(* Logix 5000 project; controller Google vendor 1 type 14 code 151 rev 31.11; software revision 31.00; part 4 of 6 *)
(* tags used below, declared in another part *)
   Elev_FWD_Delay : TIMER;
   Elev_REV_Delay : TIMER;
   Elev_Slow : BOOL;
   FaultResetDelay : TIMER;
   HMI_AutoMode : BOOL;
   HMI_LiftJogDown : BOOL;
   HMI_LiftJogUp : BOOL;
   HMI_PB_Reset : BOOL;
   Infeed_Active : BOOL;
   Infeed_Clear : BOOL;
   Infeed_Upstream_ProdCode : DINT;
   Infeed_Upstream_ProdName : STRING;
   Infeed_Z1_MinGapTimer : TIMER;
   Infeed_Z3_MinGapTimer : TIMER;
   Infeed_Zone1 : Zone_Data;
   Infeed_Zone1_2_ProdCode : DINT;
   Infeed_Zone1_2_ProdName : STRING;
   Infeed_Zone1_FWD : BOOL;
   Infeed_Zone1_PE : BOOL;
   Infeed_Zone1_ProdCode : DINT;
   Infeed_Zone1_ProdName : STRING;
   Infeed_Zone1_REV : BOOL;
   Infeed_Zone2 : Zone_Data;
   Infeed_Zone2_3_ProdCode : DINT;
   Infeed_Zone2_3_ProdName : STRING;
   Infeed_Zone2_FWD : BOOL;
   Infeed_Zone2_PE : BOOL;
   Infeed_Zone2_ProdCode : DINT;
   Infeed_Zone2_ProdName : STRING;
   Infeed_Zone2_REV : BOOL;
   Infeed_Zone3 : Zone_Data;
   Infeed_Zone3_4_ProdCode : DINT;
   Infeed_Zone3_4_ProdName : STRING;
   Infeed_Zone3_FWD : BOOL;
   Infeed_Zone3_PE : BOOL;
   Infeed_Zone3_ProdCode : DINT;
   Infeed_Zone3_ProdName : STRING;
   Infeed_Zone3_REV : BOOL;
   Infeed_Zone4 : Zone_Data;
   Infeed_Zone4_FWD : BOOL;
   Infeed_Zone4_PE : BOOL;
   Infeed_Zone4_ProdCode : DINT;
   Infeed_Zone4_ProdName : STRING;
   Infeed_Zone4_REV : BOOL;
   Infeed_Zone_Timeout : TIMER[8];
   L1_Clear_Out : BOOL;
   L1_Empty_Delay : TIMER;
   L1_Full_Delay : TIMER;
   L1_Zone1 : Zone_Data;
   L1_Zone1_2_ProdCode : DINT;
   L1_Zone1_2_ProdName : STRING;
   L1_Zone1_FWD : BOOL;
   L1_Zone1_PE : BOOL;
   L1_Zone1_ProdCode : DINT;
   L1_Zone1_ProdName : STRING;
   L1_Zone1_REV : BOOL;
   L1_Zone2 : Zone_Data;
   L1_Zone2_3_ProdCode : DINT;
   L1_Zone2_3_ProdName : STRING;
   L1_Zone2_FWD : BOOL;
   L1_Zone2_PE : BOOL;
   L1_Zone2_ProdCode : DINT;
   L1_Zone2_ProdName : STRING;
   L1_Zone2_REV : BOOL;
   L1_Zone3 : Zone_Data;
   L1_Zone3_4_ProdCode : DINT;
   L1_Zone3_4_ProdName : STRING;
   L1_Zone3_FWD : BOOL;
   L1_Zone3_PE : BOOL;
   L1_Zone3_ProdCode : DINT;
   L1_Zone3_ProdName : STRING;
   L1_Zone3_REV : BOOL;
   L1_Zone4 : End_Zone_Data;
   L1_Zone4_FWD : BOOL;
   L1_Zone4_PE : BOOL;
   L1_Zone4_ProdCode : DINT;
   L1_Zone4_ProdName : STRING;
   L1_Zone4_REV : BOOL;
   L1_Zone_Timeout : TIMER[8];
   L2_Zone1 : Zone_Data;
   L2_Zone1_REV : BOOL;
   L3_Zone1 : Zone_Data;
   L3_Zone1_REV : BOOL;
   L4_Zone1 : Zone_Data;
   L4_Zone1_REV : BOOL;
   L5_Zone1 : Zone_Data;
   L5_Zone1_REV : BOOL;
   Level_1_Empty : BOOL;
   Level_1_Full : BOOL;
   Lift_Alarm : BOOL;
   Lift_Ascend : BOOL;
   Lift_Conv_PE1 : BOOL;
   Lift_Conv_PE2 : BOOL;
   Lift_Current_Level : DINT;
   Lift_Cycle_Counter : COUNTER;
   Lift_Descend : BOOL;
   Lift_FullSpeed : DINT;
   Lift_L1_Slow_Prox : BOOL;
   Lift_L1_Stop_Prox : BOOL;
   Lift_L2_Slow_Prox : BOOL;
   Lift_L2_Stop_Prox : BOOL;
   Lift_L3_Slow_Prox : BOOL;
   Lift_L3_Stop_Prox : BOOL;
   Lift_L4_Slow_Prox : BOOL;
   Lift_L4_Stop_Prox : BOOL;
   Lift_L5_Slow_Prox : BOOL;
   Lift_L5_Stop_Prox : BOOL;
   Lift_Required_Level : DINT;
   Lift_SlowSpeed : DINT;
   Lift_Zone : Lift_Zone_Data;
   Lift_Zone_ProdCode : DINT;
   Lift_Zone_ProdName : STRING;
   Lift_Zone_Timeout : TIMER[2];
   LiftZone_FWD : BOOL;
   LiftZone_REV : BOOL;
   LiftZoneDownstream_ProdCode : DINT;
   LiftZoneDownstream_ProdName : STRING;
   LiftZoneFWD_ResetTimer : TIMER;
   LiftZoneREV_ResetTimer : TIMER;
   LiftZoneUpstream_ProdCode : DINT;
   LiftZoneUpstream_ProdName : STRING;
   ONS : DINT[6];
   Outfeed_Active : BOOL;
   Safety_Relay_Status : BOOL;
   Sort_Number : DINT;
   System : State;
   System_State : DINT;
(* MainProgram, continued *)

ROUTINE R06_Lift_Operation   (* ladder *)
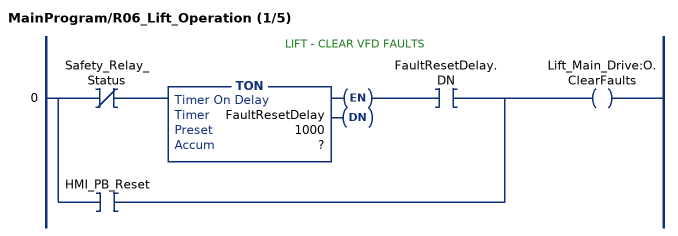
   // LIFT - CLEAR VFD FAULTS
   0: [XIO(Safety_Relay_Status) TON(FaultResetDelay,?,?) XIC(FaultResetDelay.DN) ,XIC(HMI_PB_Reset) ]OTE(Lift_Main_Drive:O.ClearFaults);
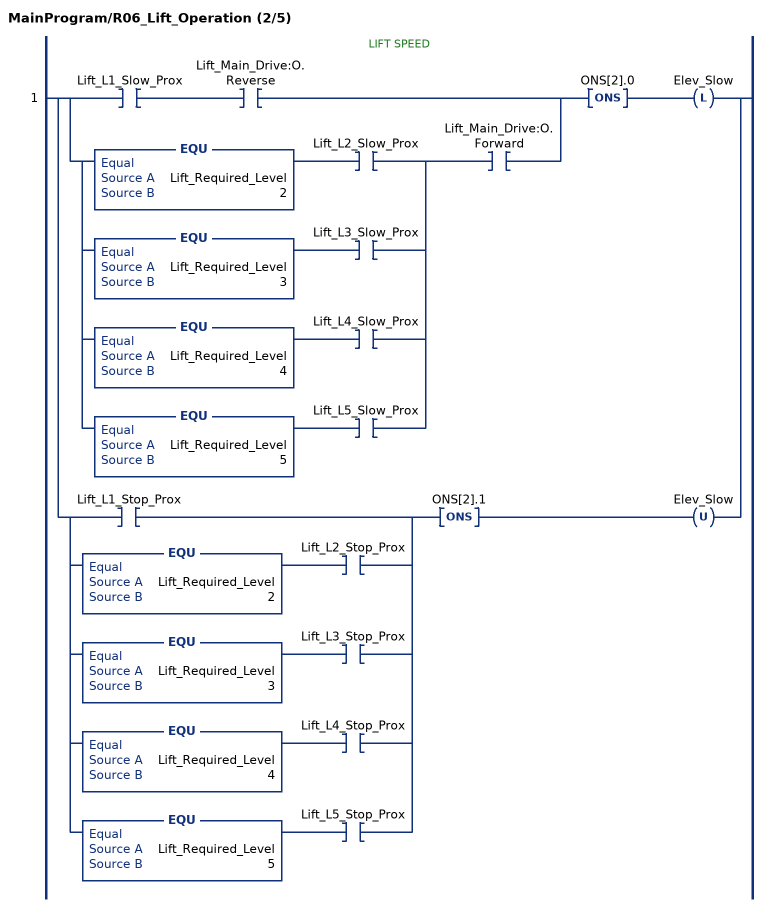
   // LIFT SPEED
   1: [[XIC(Lift_L1_Slow_Prox) XIC(Lift_Main_Drive:O.Reverse) ,[EQU(Lift_Required_Level,2) XIC(Lift_L2_Slow_Prox) ,EQU(Lift_Required_Level,3) XIC(Lift_L3_Slow_Prox) ,EQU(Lift_Required_Level,4) XIC(Lift_L4_Slow_Prox) ,EQU(Lift_Required_Level,5) XIC(Lift_L5_Slow_Prox) ] XIC(Lift_Main_Drive:O.Forward) ] ONS(ONS[2].0) OTL(Elev_Slow) ,[XIC(Lift_L1_Stop_Prox) ,EQU(Lift_Required_Level,2) XIC(Lift_L2_Stop_Prox) ,EQU(Lift_Required_Level,3) XIC(Lift_L3_Stop_Prox) ,EQU(Lift_Required_Level,4) XIC(Lift_L4_Stop_Prox) ,EQU(Lift_Required_Level,5) XIC(Lift_L5_Stop_Prox) ] ONS(ONS[2].1) OTU(Elev_Slow) ];
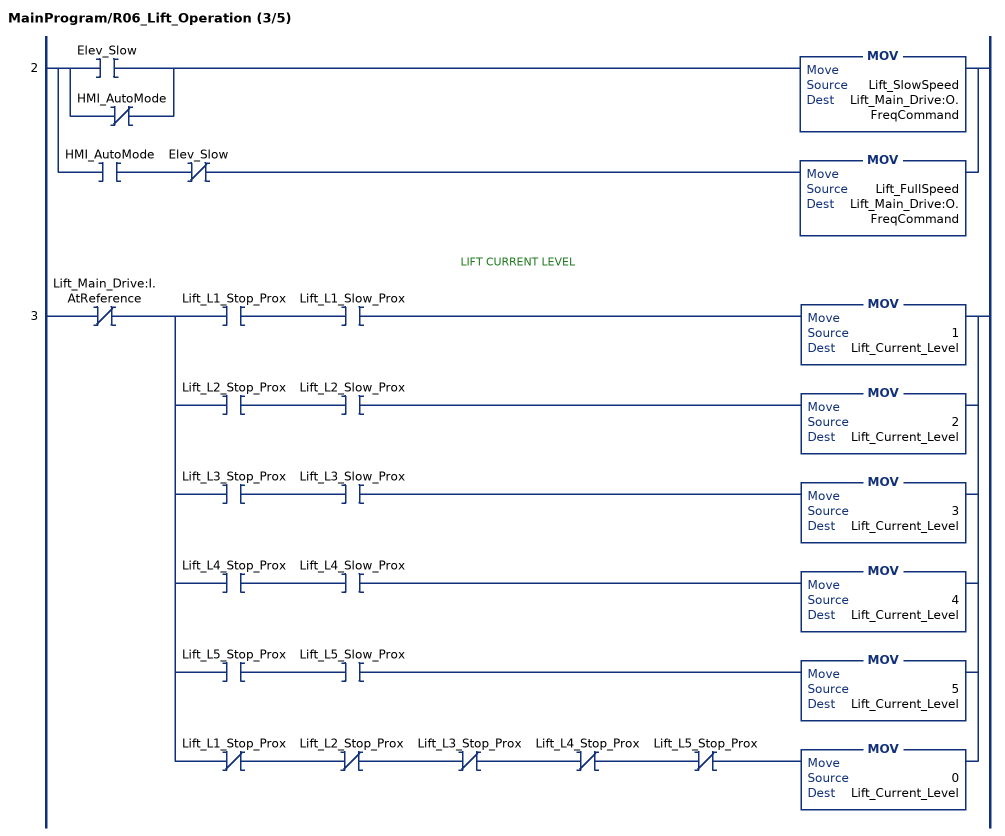
   2: [[XIC(Elev_Slow) ,XIO(HMI_AutoMode) ] MOV(Lift_SlowSpeed,Lift_Main_Drive:O.FreqCommand) ,XIC(HMI_AutoMode) XIO(Elev_Slow) MOV(Lift_FullSpeed,Lift_Main_Drive:O.FreqCommand) ];
   // LIFT CURRENT LEVEL
   3: XIO(Lift_Main_Drive:I.AtReference)[XIC(Lift_L1_Stop_Prox) XIC(Lift_L1_Slow_Prox) MOV(1,Lift_Current_Level) ,XIC(Lift_L2_Stop_Prox) XIC(Lift_L2_Slow_Prox) MOV(2,Lift_Current_Level) ,XIC(Lift_L3_Stop_Prox) XIC(Lift_L3_Slow_Prox) MOV(3,Lift_Current_Level) ,XIC(Lift_L4_Stop_Prox) XIC(Lift_L4_Slow_Prox) MOV(4,Lift_Current_Level) ,XIC(Lift_L5_Stop_Prox) XIC(Lift_L5_Slow_Prox) MOV(5,Lift_Current_Level) ,XIO(Lift_L1_Stop_Prox) XIO(Lift_L2_Stop_Prox) XIO(Lift_L3_Stop_Prox) XIO(Lift_L4_Stop_Prox) XIO(Lift_L5_Stop_Prox) MOV(0,Lift_Current_Level) ];
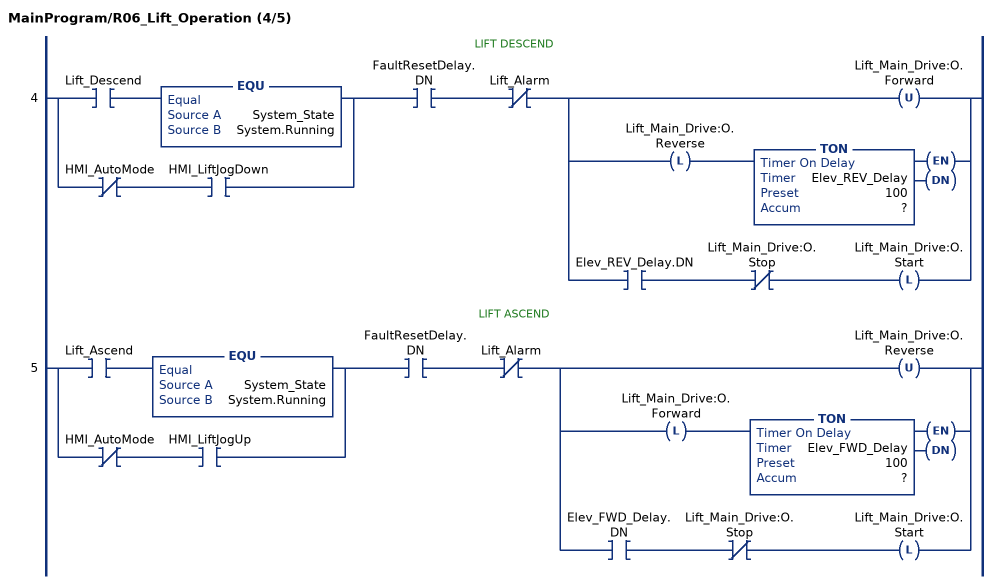
   // LIFT DESCEND
   4: [XIC(Lift_Descend) EQU(System_State,System.Running) ,XIO(HMI_AutoMode) XIC(HMI_LiftJogDown) ]XIC(FaultResetDelay.DN)XIO(Lift_Alarm)[OTU(Lift_Main_Drive:O.Forward) ,OTL(Lift_Main_Drive:O.Reverse) TON(Elev_REV_Delay,?,?) ,XIC(Elev_REV_Delay.DN) XIO(Lift_Main_Drive:O.Stop) OTL(Lift_Main_Drive:O.Start) ];
   // LIFT ASCEND
   5: [XIC(Lift_Ascend) EQU(System_State,System.Running) ,XIO(HMI_AutoMode) XIC(HMI_LiftJogUp) ]XIC(FaultResetDelay.DN)XIO(Lift_Alarm)[OTU(Lift_Main_Drive:O.Reverse) ,OTL(Lift_Main_Drive:O.Forward) TON(Elev_FWD_Delay,?,?) ,XIC(Elev_FWD_Delay.DN) XIO(Lift_Main_Drive:O.Stop) OTL(Lift_Main_Drive:O.Start) ];
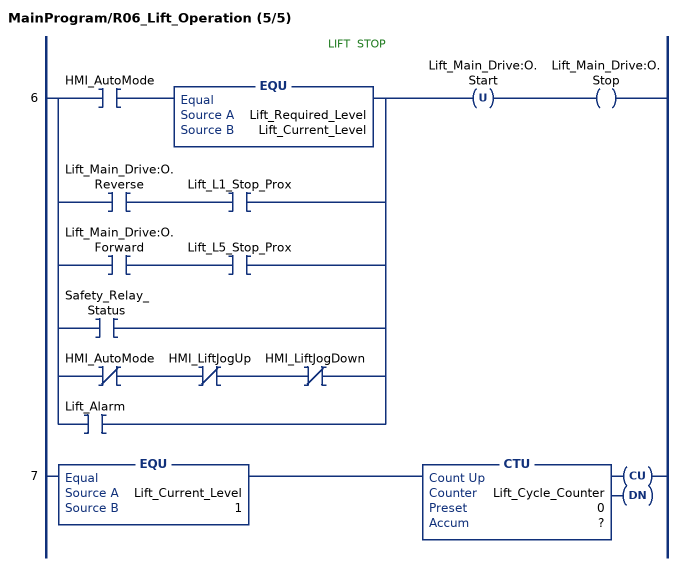
   // LIFT  STOP
   6: [XIC(HMI_AutoMode) EQU(Lift_Required_Level,Lift_Current_Level) ,XIC(Lift_Main_Drive:O.Reverse) XIC(Lift_L1_Stop_Prox) ,XIC(Lift_Main_Drive:O.Forward) XIC(Lift_L5_Stop_Prox) ,XIC(Safety_Relay_Status) ,XIO(HMI_AutoMode) XIO(HMI_LiftJogUp) XIO(HMI_LiftJogDown) ,XIC(Lift_Alarm) ]OTU(Lift_Main_Drive:O.Start)OTE(Lift_Main_Drive:O.Stop);
   7: EQU(Lift_Current_Level,1)CTU(Lift_Cycle_Counter,?,?);
END_ROUTINE

ROUTINE R07_Infeed_Conveyor   (* ladder *)
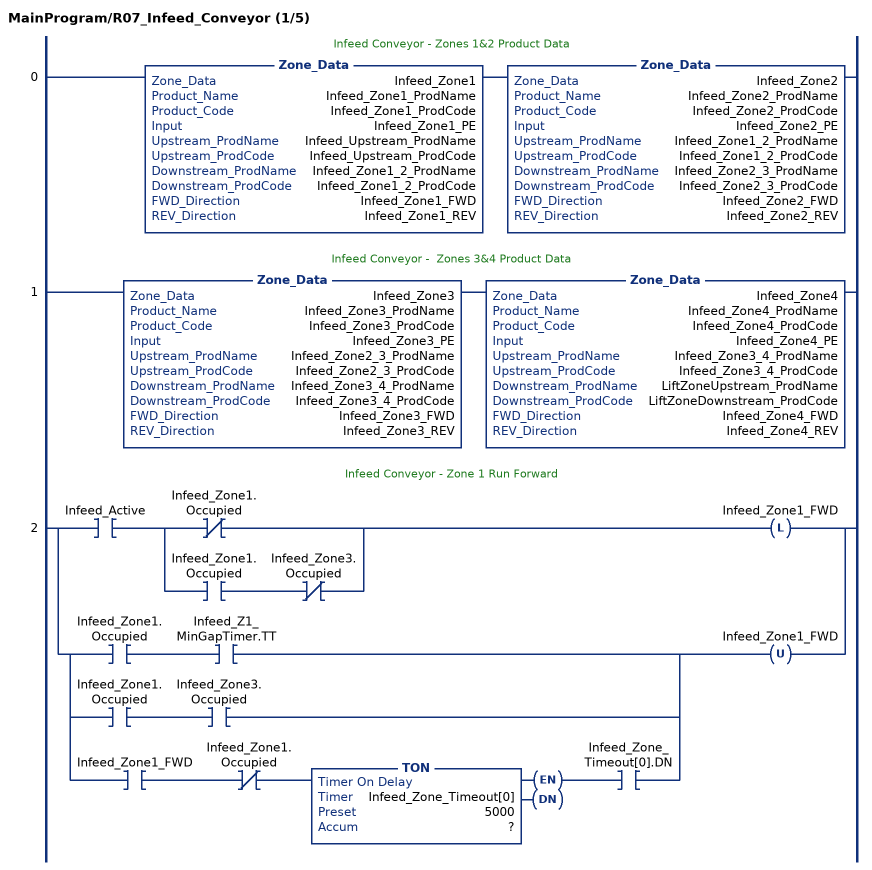
   // Infeed Conveyor - Zones 1&2 Product Data
   0: Zone_Data(Infeed_Zone1,Infeed_Zone1_ProdName,Infeed_Zone1_ProdCode,Infeed_Zone1_PE,Infeed_Upstream_ProdName,Infeed_Upstream_ProdCode,Infeed_Zone1_2_ProdName,Infeed_Zone1_2_ProdCode,Infeed_Zone1_FWD,Infeed_Zone1_REV)Zone_Data(Infeed_Zone2,Infeed_Zone2_ProdName,Infeed_Zone2_ProdCode,Infeed_Zone2_PE,Infeed_Zone1_2_ProdName,Infeed_Zone1_2_ProdCode,Infeed_Zone2_3_ProdName,Infeed_Zone2_3_ProdCode,Infeed_Zone2_FWD,Infeed_Zone2_REV);
   // Infeed Conveyor -  Zones 3&4 Product Data
   1: Zone_Data(Infeed_Zone3,Infeed_Zone3_ProdName,Infeed_Zone3_ProdCode,Infeed_Zone3_PE,Infeed_Zone2_3_ProdName,Infeed_Zone2_3_ProdCode,Infeed_Zone3_4_ProdName,Infeed_Zone3_4_ProdCode,Infeed_Zone3_FWD,Infeed_Zone3_REV)Zone_Data(Infeed_Zone4,Infeed_Zone4_ProdName,Infeed_Zone4_ProdCode,Infeed_Zone4_PE,Infeed_Zone3_4_ProdName,Infeed_Zone3_4_ProdCode,LiftZoneUpstream_ProdName,LiftZoneDownstream_ProdCode,Infeed_Zone4_FWD,Infeed_Zone4_REV);
   // Infeed Conveyor - Zone 1 Run Forward
   2: [XIC(Infeed_Active) [XIO(Infeed_Zone1.Occupied) ,XIC(Infeed_Zone1.Occupied) XIO(Infeed_Zone3.Occupied) ] OTL(Infeed_Zone1_FWD) ,[XIC(Infeed_Zone1.Occupied) XIC(Infeed_Z1_MinGapTimer.TT) ,XIC(Infeed_Zone1.Occupied) XIC(Infeed_Zone3.Occupied) ,XIC(Infeed_Zone1_FWD) XIO(Infeed_Zone1.Occupied) TON(Infeed_Zone_Timeout[0],?,?) XIC(Infeed_Zone_Timeout[0].DN) ] OTU(Infeed_Zone1_FWD) ];
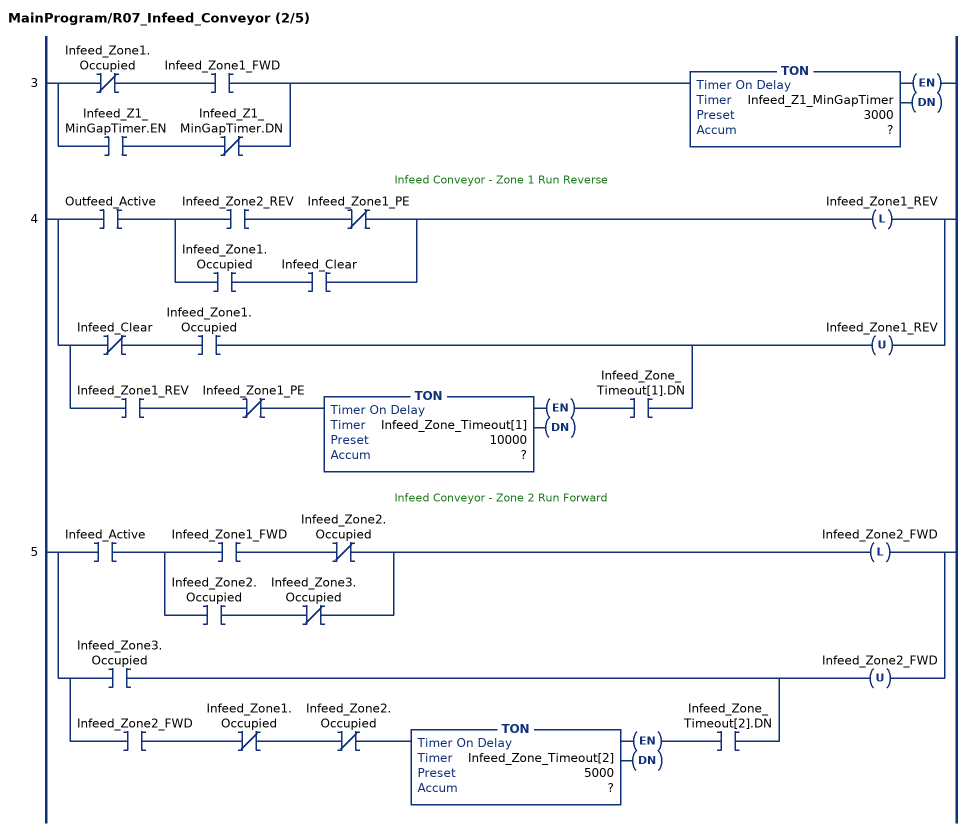
   3: [XIO(Infeed_Zone1.Occupied) XIC(Infeed_Zone1_FWD) ,XIC(Infeed_Z1_MinGapTimer.EN) XIO(Infeed_Z1_MinGapTimer.DN) ]TON(Infeed_Z1_MinGapTimer,?,?);
   // Infeed Conveyor - Zone 1 Run Reverse
   4: [XIC(Outfeed_Active) [XIC(Infeed_Zone2_REV) XIO(Infeed_Zone1_PE) ,XIC(Infeed_Zone1.Occupied) XIC(Infeed_Clear) ] OTL(Infeed_Zone1_REV) ,[XIO(Infeed_Clear) XIC(Infeed_Zone1.Occupied) ,XIC(Infeed_Zone1_REV) XIO(Infeed_Zone1_PE) TON(Infeed_Zone_Timeout[1],?,?) XIC(Infeed_Zone_Timeout[1].DN) ] OTU(Infeed_Zone1_REV) ];
   // Infeed Conveyor - Zone 2 Run Forward
   5: [XIC(Infeed_Active) [XIC(Infeed_Zone1_FWD) XIO(Infeed_Zone2.Occupied) ,XIC(Infeed_Zone2.Occupied) XIO(Infeed_Zone3.Occupied) ] OTL(Infeed_Zone2_FWD) ,[XIC(Infeed_Zone3.Occupied) ,XIC(Infeed_Zone2_FWD) XIO(Infeed_Zone1.Occupied) XIO(Infeed_Zone2.Occupied) TON(Infeed_Zone_Timeout[2],?,?) XIC(Infeed_Zone_Timeout[2].DN) ] OTU(Infeed_Zone2_FWD) ];
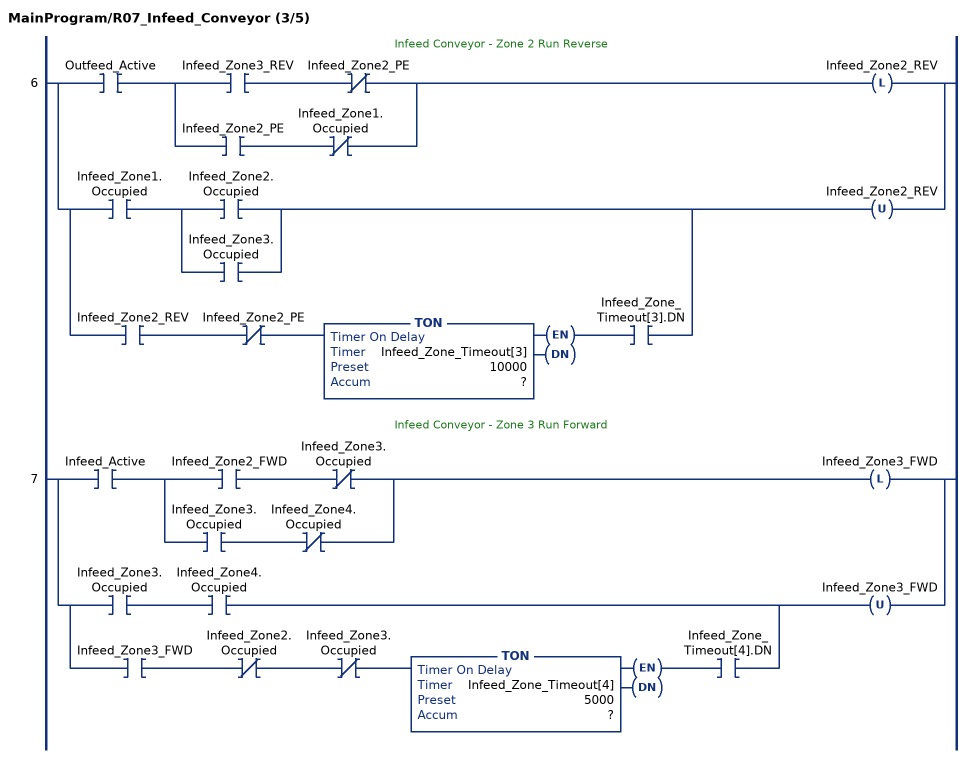
   // Infeed Conveyor - Zone 2 Run Reverse
   6: [XIC(Outfeed_Active) [XIC(Infeed_Zone3_REV) XIO(Infeed_Zone2_PE) ,XIC(Infeed_Zone2_PE) XIO(Infeed_Zone1.Occupied) ] OTL(Infeed_Zone2_REV) ,[XIC(Infeed_Zone1.Occupied) [XIC(Infeed_Zone2.Occupied) ,XIC(Infeed_Zone3.Occupied) ] ,XIC(Infeed_Zone2_REV) XIO(Infeed_Zone2_PE) TON(Infeed_Zone_Timeout[3],?,?) XIC(Infeed_Zone_Timeout[3].DN) ] OTU(Infeed_Zone2_REV) ];
   // Infeed Conveyor - Zone 3 Run Forward
   7: [XIC(Infeed_Active) [XIC(Infeed_Zone2_FWD) XIO(Infeed_Zone3.Occupied) ,XIC(Infeed_Zone3.Occupied) XIO(Infeed_Zone4.Occupied) ] OTL(Infeed_Zone3_FWD) ,[XIC(Infeed_Zone3.Occupied) XIC(Infeed_Zone4.Occupied) ,XIC(Infeed_Zone3_FWD) XIO(Infeed_Zone2.Occupied) XIO(Infeed_Zone3.Occupied) TON(Infeed_Zone_Timeout[4],?,?) XIC(Infeed_Zone_Timeout[4].DN) ] OTU(Infeed_Zone3_FWD) ];
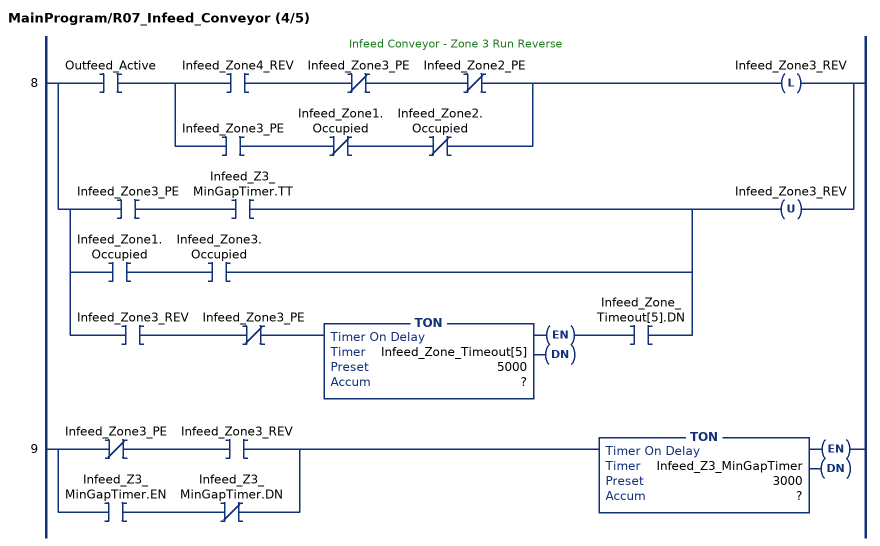
   // Infeed Conveyor - Zone 3 Run Reverse
   8: [XIC(Outfeed_Active) [XIC(Infeed_Zone4_REV) XIO(Infeed_Zone3_PE) XIO(Infeed_Zone2_PE) ,XIC(Infeed_Zone3_PE) XIO(Infeed_Zone1.Occupied) XIO(Infeed_Zone2.Occupied) ] OTL(Infeed_Zone3_REV) ,[XIC(Infeed_Zone3_PE) XIC(Infeed_Z3_MinGapTimer.TT) ,XIC(Infeed_Zone1.Occupied) XIC(Infeed_Zone3.Occupied) ,XIC(Infeed_Zone3_REV) XIO(Infeed_Zone3_PE) TON(Infeed_Zone_Timeout[5],?,?) XIC(Infeed_Zone_Timeout[5].DN) ] OTU(Infeed_Zone3_REV) ];
   9: [XIO(Infeed_Zone3_PE) XIC(Infeed_Zone3_REV) ,XIC(Infeed_Z3_MinGapTimer.EN) XIO(Infeed_Z3_MinGapTimer.DN) ]TON(Infeed_Z3_MinGapTimer,?,?);
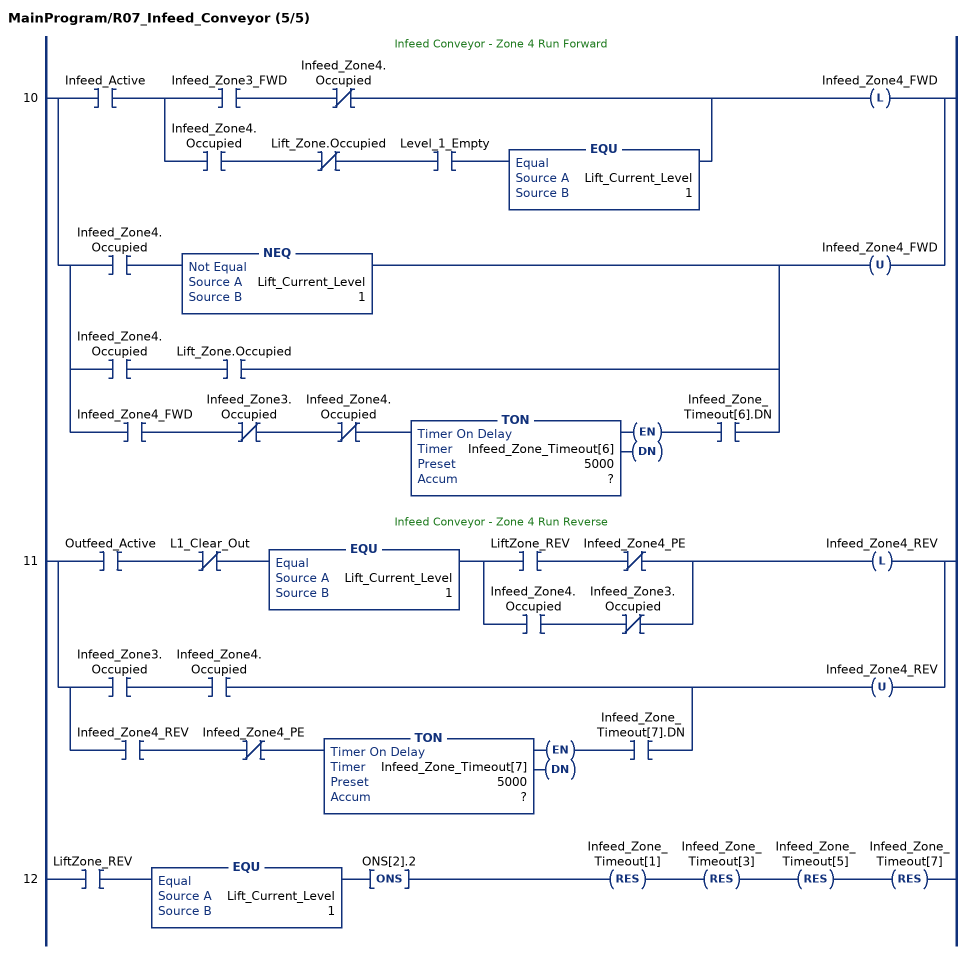
   // Infeed Conveyor - Zone 4 Run Forward
   10: [XIC(Infeed_Active) [XIC(Infeed_Zone3_FWD) XIO(Infeed_Zone4.Occupied) ,XIC(Infeed_Zone4.Occupied) XIO(Lift_Zone.Occupied) XIC(Level_1_Empty) EQU(Lift_Current_Level,1) ] OTL(Infeed_Zone4_FWD) ,[XIC(Infeed_Zone4.Occupied) NEQ(Lift_Current_Level,1) ,XIC(Infeed_Zone4.Occupied) XIC(Lift_Zone.Occupied) ,XIC(Infeed_Zone4_FWD) XIO(Infeed_Zone3.Occupied) XIO(Infeed_Zone4.Occupied) TON(Infeed_Zone_Timeout[6],?,?) XIC(Infeed_Zone_Timeout[6].DN) ] OTU(Infeed_Zone4_FWD) ];
   // Infeed Conveyor - Zone 4 Run Reverse
   11: [XIC(Outfeed_Active) XIO(L1_Clear_Out) EQU(Lift_Current_Level,1) [XIC(LiftZone_REV) XIO(Infeed_Zone4_PE) ,XIC(Infeed_Zone4.Occupied) XIO(Infeed_Zone3.Occupied) ] OTL(Infeed_Zone4_REV) ,[XIC(Infeed_Zone3.Occupied) XIC(Infeed_Zone4.Occupied) ,XIC(Infeed_Zone4_REV) XIO(Infeed_Zone4_PE) TON(Infeed_Zone_Timeout[7],?,?) XIC(Infeed_Zone_Timeout[7].DN) ] OTU(Infeed_Zone4_REV) ];
   12: XIC(LiftZone_REV)EQU(Lift_Current_Level,1)ONS(ONS[2].2)RES(Infeed_Zone_Timeout[1])RES(Infeed_Zone_Timeout[3])RES(Infeed_Zone_Timeout[5])RES(Infeed_Zone_Timeout[7]);
END_ROUTINE

ROUTINE R08_Lift_Conveyor   (* ladder *)
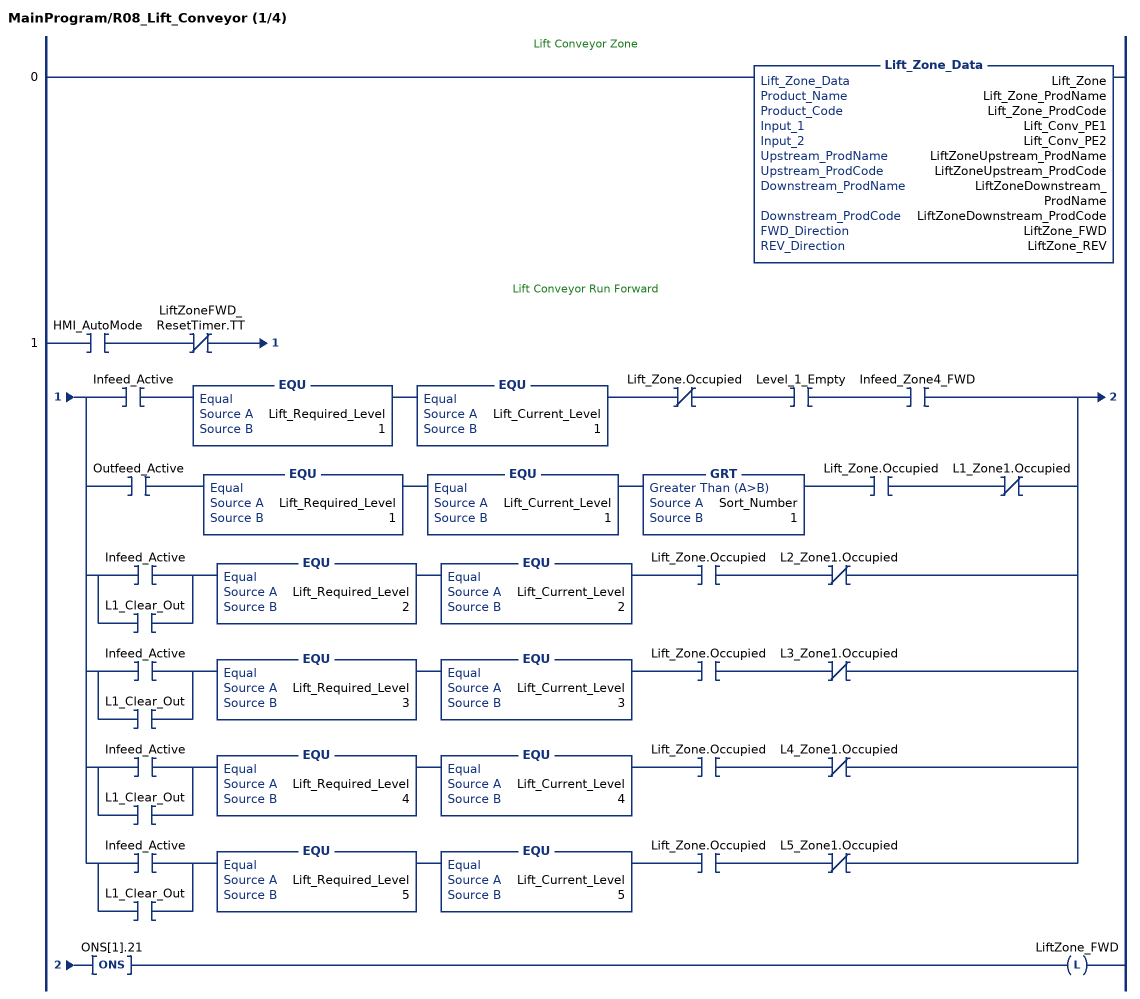
   // Lift Conveyor Zone
   0: Lift_Zone_Data(Lift_Zone,Lift_Zone_ProdName,Lift_Zone_ProdCode,Lift_Conv_PE1,Lift_Conv_PE2,LiftZoneUpstream_ProdName,LiftZoneUpstream_ProdCode,LiftZoneDownstream_ProdName,LiftZoneDownstream_ProdCode,LiftZone_FWD,LiftZone_REV);
   // Lift Conveyor Run Forward
   1: XIC(HMI_AutoMode)XIO(LiftZoneFWD_ResetTimer.TT)[XIC(Infeed_Active) EQU(Lift_Required_Level,1) EQU(Lift_Current_Level,1) XIO(Lift_Zone.Occupied) XIC(Level_1_Empty) XIC(Infeed_Zone4_FWD) ,XIC(Outfeed_Active) EQU(Lift_Required_Level,1) EQU(Lift_Current_Level,1) GRT(Sort_Number,1) XIC(Lift_Zone.Occupied) XIO(L1_Zone1.Occupied) ,[XIC(Infeed_Active) ,XIC(L1_Clear_Out) ] EQU(Lift_Required_Level,2) EQU(Lift_Current_Level,2) XIC(Lift_Zone.Occupied) XIO(L2_Zone1.Occupied) ,[XIC(Infeed_Active) ,XIC(L1_Clear_Out) ] EQU(Lift_Required_Level,3) EQU(Lift_Current_Level,3) XIC(Lift_Zone.Occupied) XIO(L3_Zone1.Occupied) ,[XIC(Infeed_Active) ,XIC(L1_Clear_Out) ] EQU(Lift_Required_Level,4) EQU(Lift_Current_Level,4) XIC(Lift_Zone.Occupied) XIO(L4_Zone1.Occupied) ,[XIC(Infeed_Active) ,XIC(L1_Clear_Out) ] EQU(Lift_Required_Level,5) EQU(Lift_Current_Level,5) XIC(Lift_Zone.Occupied) XIO(L5_Zone1.Occupied) ]ONS(ONS[1].21)OTL(LiftZone_FWD);
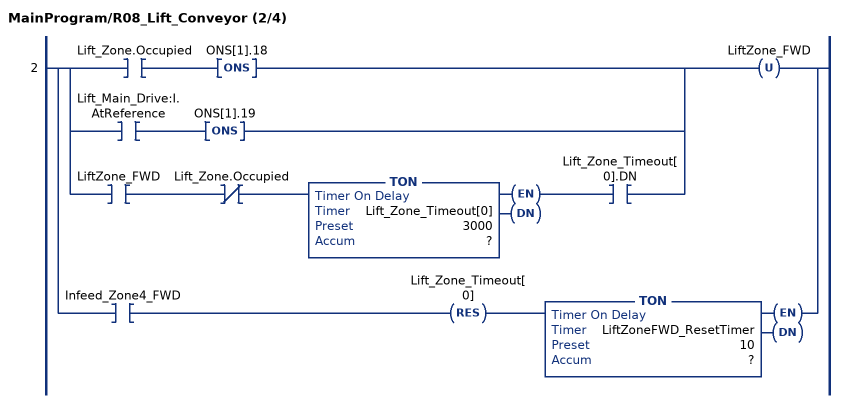
   2: [[XIC(Lift_Zone.Occupied) ONS(ONS[1].18) ,XIC(Lift_Main_Drive:I.AtReference) ONS(ONS[1].19) ,XIC(LiftZone_FWD) XIO(Lift_Zone.Occupied) TON(Lift_Zone_Timeout[0],?,?) XIC(Lift_Zone_Timeout[0].DN) ] OTU(LiftZone_FWD) ,XIC(Infeed_Zone4_FWD) RES(Lift_Zone_Timeout[0]) TON(LiftZoneFWD_ResetTimer,?,?) ];
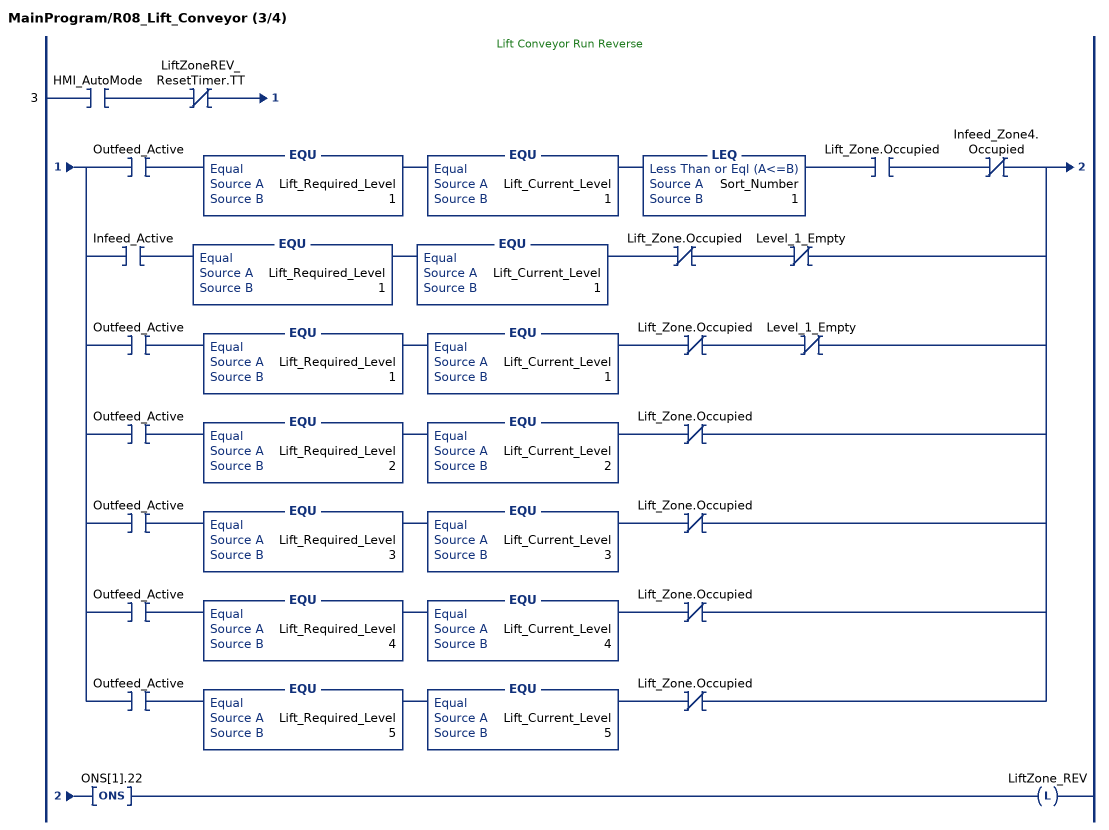
   // Lift Conveyor Run Reverse
   3: XIC(HMI_AutoMode)XIO(LiftZoneREV_ResetTimer.TT)[XIC(Outfeed_Active) EQU(Lift_Required_Level,1) EQU(Lift_Current_Level,1) LEQ(Sort_Number,1) XIC(Lift_Zone.Occupied) XIO(Infeed_Zone4.Occupied) ,XIC(Infeed_Active) EQU(Lift_Required_Level,1) EQU(Lift_Current_Level,1) XIO(Lift_Zone.Occupied) XIO(Level_1_Empty) ,XIC(Outfeed_Active) EQU(Lift_Required_Level,1) EQU(Lift_Current_Level,1) XIO(Lift_Zone.Occupied) XIO(Level_1_Empty) ,XIC(Outfeed_Active) EQU(Lift_Required_Level,2) EQU(Lift_Current_Level,2) XIO(Lift_Zone.Occupied) ,XIC(Outfeed_Active) EQU(Lift_Required_Level,3) EQU(Lift_Current_Level,3) XIO(Lift_Zone.Occupied) ,XIC(Outfeed_Active) EQU(Lift_Required_Level,4) EQU(Lift_Current_Level,4) XIO(Lift_Zone.Occupied) ,XIC(Outfeed_Active) EQU(Lift_Required_Level,5) EQU(Lift_Current_Level,5) XIO(Lift_Zone.Occupied) ]ONS(ONS[1].22)OTL(LiftZone_REV);
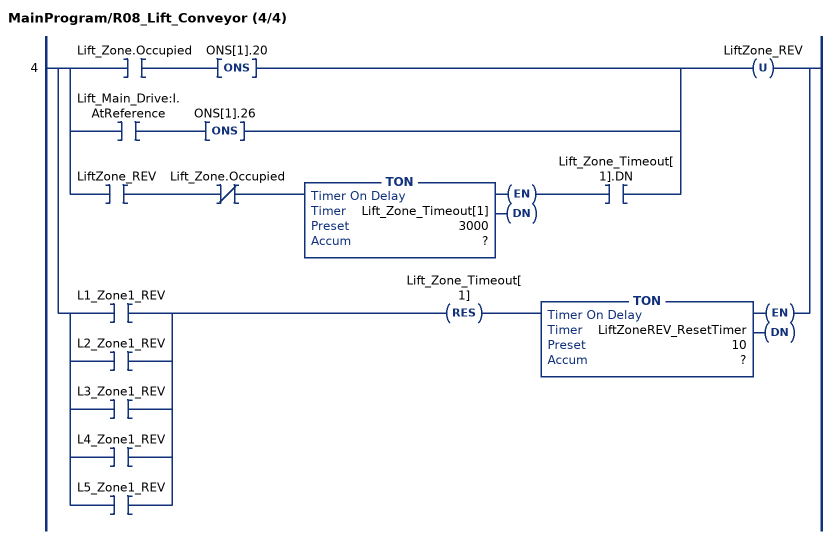
   4: [[XIC(Lift_Zone.Occupied) ONS(ONS[1].20) ,XIC(Lift_Main_Drive:I.AtReference) ONS(ONS[1].26) ,XIC(LiftZone_REV) XIO(Lift_Zone.Occupied) TON(Lift_Zone_Timeout[1],?,?) XIC(Lift_Zone_Timeout[1].DN) ] OTU(LiftZone_REV) ,[XIC(L1_Zone1_REV) ,XIC(L2_Zone1_REV) ,XIC(L3_Zone1_REV) ,XIC(L4_Zone1_REV) ,XIC(L5_Zone1_REV) ] RES(Lift_Zone_Timeout[1]) TON(LiftZoneREV_ResetTimer,?,?) ];
END_ROUTINE

ROUTINE R09_L1_Conveyor   (* ladder *)
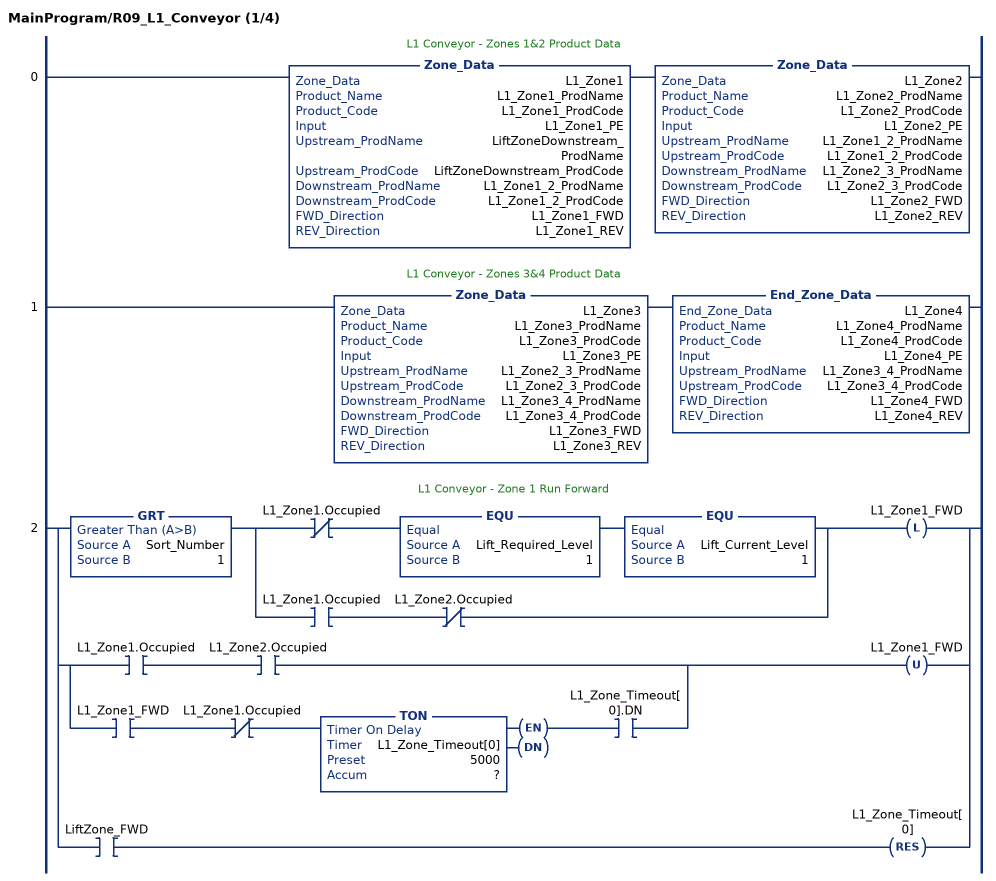
   // L1 Conveyor - Zones 1&2 Product Data
   0: Zone_Data(L1_Zone1,L1_Zone1_ProdName,L1_Zone1_ProdCode,L1_Zone1_PE,LiftZoneDownstream_ProdName,LiftZoneDownstream_ProdCode,L1_Zone1_2_ProdName,L1_Zone1_2_ProdCode,L1_Zone1_FWD,L1_Zone1_REV)Zone_Data(L1_Zone2,L1_Zone2_ProdName,L1_Zone2_ProdCode,L1_Zone2_PE,L1_Zone1_2_ProdName,L1_Zone1_2_ProdCode,L1_Zone2_3_ProdName,L1_Zone2_3_ProdCode,L1_Zone2_FWD,L1_Zone2_REV);
   // L1 Conveyor - Zones 3&4 Product Data
   1: Zone_Data(L1_Zone3,L1_Zone3_ProdName,L1_Zone3_ProdCode,L1_Zone3_PE,L1_Zone2_3_ProdName,L1_Zone2_3_ProdCode,L1_Zone3_4_ProdName,L1_Zone3_4_ProdCode,L1_Zone3_FWD,L1_Zone3_REV)End_Zone_Data(L1_Zone4,L1_Zone4_ProdName,L1_Zone4_ProdCode,L1_Zone4_PE,L1_Zone3_4_ProdName,L1_Zone3_4_ProdCode,L1_Zone4_FWD,L1_Zone4_REV);
   // L1 Conveyor - Zone 1 Run Forward
   2: [GRT(Sort_Number,1) [XIO(L1_Zone1.Occupied) EQU(Lift_Required_Level,1) EQU(Lift_Current_Level,1) ,XIC(L1_Zone1.Occupied) XIO(L1_Zone2.Occupied) ] OTL(L1_Zone1_FWD) ,[XIC(L1_Zone1.Occupied) XIC(L1_Zone2.Occupied) ,XIC(L1_Zone1_FWD) XIO(L1_Zone1.Occupied) TON(L1_Zone_Timeout[0],?,?) XIC(L1_Zone_Timeout[0].DN) ] OTU(L1_Zone1_FWD) ,XIC(LiftZone_FWD) RES(L1_Zone_Timeout[0]) ];
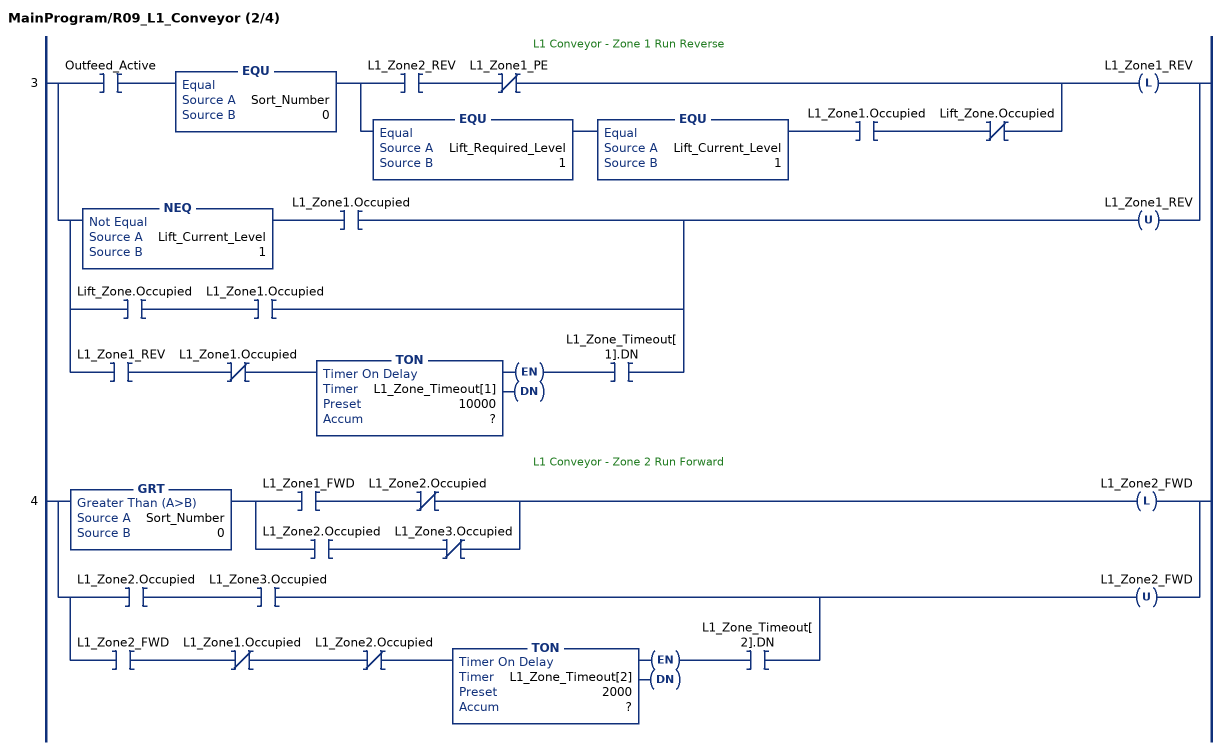
   // L1 Conveyor - Zone 1 Run Reverse
   3: [XIC(Outfeed_Active) EQU(Sort_Number,0) [XIC(L1_Zone2_REV) XIO(L1_Zone1_PE) ,EQU(Lift_Required_Level,1) EQU(Lift_Current_Level,1) XIC(L1_Zone1.Occupied) XIO(Lift_Zone.Occupied) ] OTL(L1_Zone1_REV) ,[NEQ(Lift_Current_Level,1) XIC(L1_Zone1.Occupied) ,XIC(Lift_Zone.Occupied) XIC(L1_Zone1.Occupied) ,XIC(L1_Zone1_REV) XIO(L1_Zone1.Occupied) TON(L1_Zone_Timeout[1],?,?) XIC(L1_Zone_Timeout[1].DN) ] OTU(L1_Zone1_REV) ];
   // L1 Conveyor - Zone 2 Run Forward
   4: [GRT(Sort_Number,0) [XIC(L1_Zone1_FWD) XIO(L1_Zone2.Occupied) ,XIC(L1_Zone2.Occupied) XIO(L1_Zone3.Occupied) ] OTL(L1_Zone2_FWD) ,[XIC(L1_Zone2.Occupied) XIC(L1_Zone3.Occupied) ,XIC(L1_Zone2_FWD) XIO(L1_Zone1.Occupied) XIO(L1_Zone2.Occupied) TON(L1_Zone_Timeout[2],?,?) XIC(L1_Zone_Timeout[2].DN) ] OTU(L1_Zone2_FWD) ];
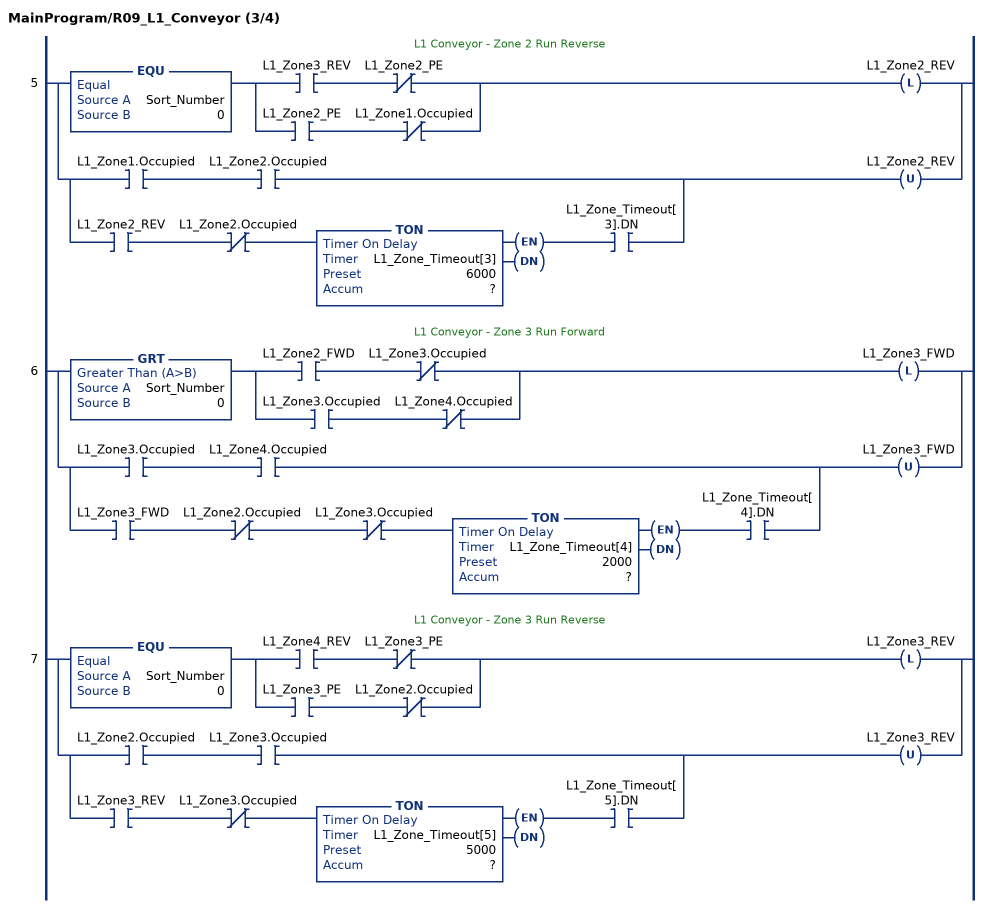
   // L1 Conveyor - Zone 2 Run Reverse
   5: [EQU(Sort_Number,0) [XIC(L1_Zone3_REV) XIO(L1_Zone2_PE) ,XIC(L1_Zone2_PE) XIO(L1_Zone1.Occupied) ] OTL(L1_Zone2_REV) ,[XIC(L1_Zone1.Occupied) XIC(L1_Zone2.Occupied) ,XIC(L1_Zone2_REV) XIO(L1_Zone2.Occupied) TON(L1_Zone_Timeout[3],?,?) XIC(L1_Zone_Timeout[3].DN) ] OTU(L1_Zone2_REV) ];
   // L1 Conveyor - Zone 3 Run Forward
   6: [GRT(Sort_Number,0) [XIC(L1_Zone2_FWD) XIO(L1_Zone3.Occupied) ,XIC(L1_Zone3.Occupied) XIO(L1_Zone4.Occupied) ] OTL(L1_Zone3_FWD) ,[XIC(L1_Zone3.Occupied) XIC(L1_Zone4.Occupied) ,XIC(L1_Zone3_FWD) XIO(L1_Zone2.Occupied) XIO(L1_Zone3.Occupied) TON(L1_Zone_Timeout[4],?,?) XIC(L1_Zone_Timeout[4].DN) ] OTU(L1_Zone3_FWD) ];
   // L1 Conveyor - Zone 3 Run Reverse
   7: [EQU(Sort_Number,0) [XIC(L1_Zone4_REV) XIO(L1_Zone3_PE) ,XIC(L1_Zone3_PE) XIO(L1_Zone2.Occupied) ] OTL(L1_Zone3_REV) ,[XIC(L1_Zone2.Occupied) XIC(L1_Zone3.Occupied) ,XIC(L1_Zone3_REV) XIO(L1_Zone3.Occupied) TON(L1_Zone_Timeout[5],?,?) XIC(L1_Zone_Timeout[5].DN) ] OTU(L1_Zone3_REV) ];
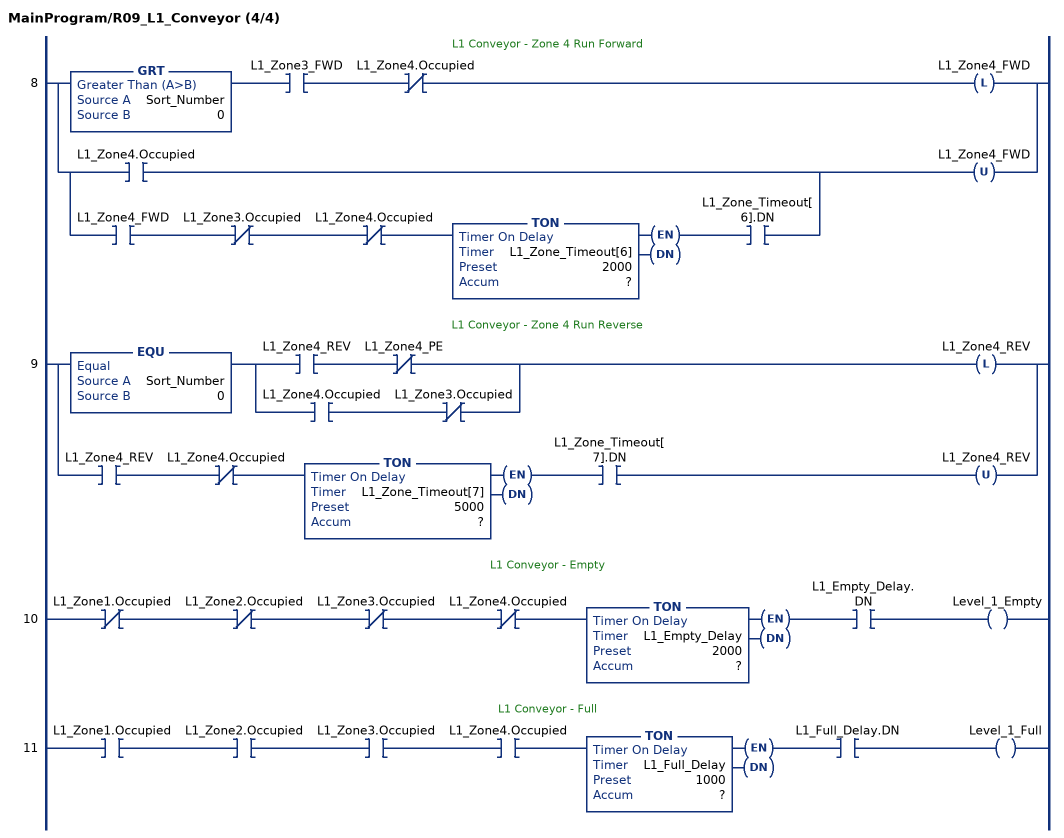
   // L1 Conveyor - Zone 4 Run Forward
   8: [GRT(Sort_Number,0) XIC(L1_Zone3_FWD) XIO(L1_Zone4.Occupied) OTL(L1_Zone4_FWD) ,[XIC(L1_Zone4.Occupied) ,XIC(L1_Zone4_FWD) XIO(L1_Zone3.Occupied) XIO(L1_Zone4.Occupied) TON(L1_Zone_Timeout[6],?,?) XIC(L1_Zone_Timeout[6].DN) ] OTU(L1_Zone4_FWD) ];
   // L1 Conveyor - Zone 4 Run Reverse
   9: [EQU(Sort_Number,0) [XIC(L1_Zone4_REV) XIO(L1_Zone4_PE) ,XIC(L1_Zone4.Occupied) XIO(L1_Zone3.Occupied) ] OTL(L1_Zone4_REV) ,XIC(L1_Zone4_REV) XIO(L1_Zone4.Occupied) TON(L1_Zone_Timeout[7],?,?) XIC(L1_Zone_Timeout[7].DN) OTU(L1_Zone4_REV) ];
   // L1 Conveyor - Empty
   10: XIO(L1_Zone1.Occupied)XIO(L1_Zone2.Occupied)XIO(L1_Zone3.Occupied)XIO(L1_Zone4.Occupied)TON(L1_Empty_Delay,?,?)XIC(L1_Empty_Delay.DN)OTE(Level_1_Empty);
   // L1 Conveyor - Full
   11: XIC(L1_Zone1.Occupied)XIC(L1_Zone2.Occupied)XIC(L1_Zone3.Occupied)XIC(L1_Zone4.Occupied)TON(L1_Full_Delay,?,?)XIC(L1_Full_Delay.DN)OTE(Level_1_Full);
END_ROUTINE
